(* PLC project fourwaytrafficlight, Unknown Unnamed 1 *)
(* stored: creationDateTime 2023-03-05T04:05:10, modificationDateTime 2023-03-16T22:44:41 *)

(* 4waytrafficlight *)
PROGRAM TRAFFICLIGHTS
  VAR
    ACTG : BOOL;  (* A and C turn Green *)
  END_VAR
  VAR_INPUT
    ACT : BOOL := 1;  (* sensor for cars in the A and C turning lane *)
  END_VAR
  VAR
    ACTY : BOOL;  (* A and C turn Yellow *)
    ACTR : BOOL;  (* A and C turn Red *)
    ACSG : BOOL;  (* A and C Straight Green *)
    ACSY : BOOL;  (* A and C Straight Yellow *)
    ACSR : BOOL;  (* A and C Straight Red *)
    BDTG : BOOL;  (* B and D Turn Green *)
    BDTY : BOOL;  (* B and D Turn Yellow *)
  END_VAR
  VAR_INPUT
    PB0 : BOOL := 1;  (* System On Switch *)
  END_VAR
  VAR
    BDTR : BOOL;  (* B and D Turn Red *)
    BDSG : BOOL;  (* B and D Straight Green *)
    BDSY : BOOL;  (* B and D Straight Yellow *)
    BDSR : BOOL;  (* B and D Straight Red *)
    TP0 : TP;
    F_TRIG1 : F_TRIG;
    TP2 : TP;
    F_TRIG2 : F_TRIG;
    R_TRIG1 : R_TRIG;
    TP3 : TP;
    F_TRIG4 : F_TRIG;
    TP4 : TP;
    F_TRIG5 : F_TRIG;
    R_TRIG2 : R_TRIG;
    TP6 : TP;
    F_TRIG7 : F_TRIG;
    TP7 : TP;
    F_TRIG8 : F_TRIG;
    R_TRIG4 : R_TRIG;
    TP9 : TP;
    F_TRIG10 : F_TRIG;
    TP10 : TP;
    F_TRIG11 : F_TRIG;
    R_TRIG3 : R_TRIG;
    R_TRIG0 : R_TRIG;
    RS0 : RS;
    RS1 : RS;
    RS2 : RS;
    RS3 : RS;
    TP1 : TP;
  END_VAR
  VAR  (* added by the conversion: wires and edge detectors of the diagram *)
    _OR25_OUT : BOOL;
  END_VAR

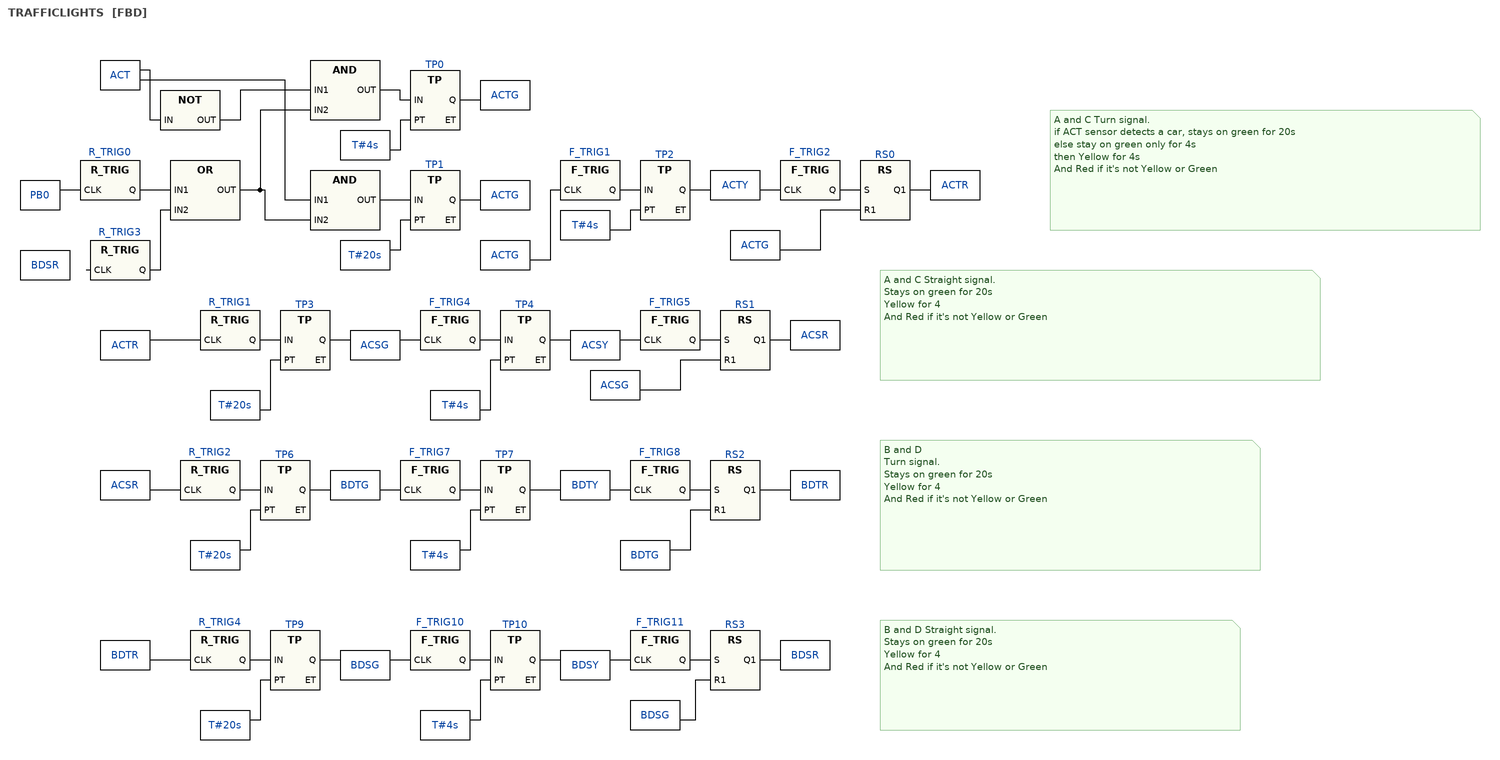
(* FBD diagram, written out as Structured Text *)
R_TRIG0(CLK := PB0);
R_TRIG3(CLK := BDSR);
_OR25_OUT := R_TRIG0.Q OR R_TRIG3.Q;
TP0(IN := NOT ACT AND _OR25_OUT, PT := T#4s);
ACTG := TP0.Q;
(* A and C Turn signal.
if ACT sensor detects a car, stays on green for 20s
   else stay on green only for 4s
then Yellow for 4s
And Red if it's not Yellow or Green *)
F_TRIG1(CLK := ACTG);
TP2(IN := F_TRIG1.Q, PT := T#4s);
ACTY := TP2.Q;
F_TRIG2(CLK := ACTY);
RS0(S := F_TRIG2.Q, R1 := ACTG);
ACTR := RS0.Q1;
TP1(IN := ACT AND _OR25_OUT, PT := T#20s);
ACTG := TP1.Q;
(* A and C Straight signal.
Stays on green for 20s
Yellow for 4
And Red if it's not Yellow or Green *)
F_TRIG5(CLK := ACSY);
RS1(S := F_TRIG5.Q, R1 := ACSG);
ACSR := RS1.Q1;
R_TRIG1(CLK := ACTR);
TP3(IN := R_TRIG1.Q, PT := T#20s);
ACSG := TP3.Q;
F_TRIG4(CLK := ACSG);
TP4(IN := F_TRIG4.Q, PT := T#4s);
ACSY := TP4.Q;
(* B and D
 Turn signal.
Stays on green for 20s
Yellow for 4
And Red if it's not Yellow or Green *)
R_TRIG2(CLK := ACSR);
TP6(IN := R_TRIG2.Q, PT := T#20s);
BDTG := TP6.Q;
F_TRIG7(CLK := BDTG);
TP7(IN := F_TRIG7.Q, PT := T#4s);
BDTY := TP7.Q;
F_TRIG8(CLK := BDTY);
RS2(S := F_TRIG8.Q, R1 := BDTG);
BDTR := RS2.Q1;
(* B and D Straight signal.
Stays on green for 20s
Yellow for 4
And Red if it's not Yellow or Green *)
F_TRIG11(CLK := BDSY);
RS3(S := F_TRIG11.Q, R1 := BDSG);
BDSR := RS3.Q1;
R_TRIG4(CLK := BDTR);
TP9(IN := R_TRIG4.Q, PT := T#20s);
BDSG := TP9.Q;
F_TRIG10(CLK := BDSG);
TP10(IN := F_TRIG10.Q, PT := T#4s);
BDSY := TP10.Q;
END_PROGRAM

CONFIGURATION Config0
  RESOURCE Res0 ON PLC
    TASK task0(INTERVAL := T#20ms, PRIORITY := 0);
    PROGRAM instance0 WITH task0 : TRAFFICLIGHTS;
  END_RESOURCE
END_CONFIGURATION
